PROGRAM MobjectDeserializationUnitTests
VAR
	deserializerGarbageCollector_TestSuite : DeserializerGarbageCollector_TestSuite;
	missingKeyDeserializationError_TestSuite :MissingKeyDeserializationError_TestSuite;
	invalidKeyDeserializationError_TestSuite : InvalidKeyDeserializationError_TestSuite;
	incorrectTypeDeserializationError_TestSuite : IncorrectTypeDeserializationError_TestSuite;
	incorrectKeyTypeDeserializationError_TestSuite : IncorrectKeyTypeDeserializationError_TestSuite;
	deserializationErrorFactory_TestSuite : DeserializationErrorFactory_TestSuite;
	customDeserializationFailedError_TestSuite : CustomDeserializationFailedError_TestSuite;
END_VAR

END_PROGRAM

(* stored: Version 1.1.0.1, ProductVersion 3.1.4024.12
   POU MobjectDeserializationUnitTests: Id {c70500cf-7d23-0663-1d50-284054be19c0}, SpecialFunc None *)
